{attribute 'qualified_only'}
{attribute 'strict'}
TYPE E_UserMgmtEventType :
(
	None := 0,
    UserCreated := 1,
    UserDeleted := 2,
    GroupUpdated := 3,
    AutoLogoutUpdated := 4,
    UserUpdated := 5,
    PasswordChanged := 6
);
END_TYPE

(* stored: Version 1.1.0.1, ProductVersion 3.1.4024.15
   DUT E_UserMgmtEventType: Id {1c1d8daf-4605-42b1-8235-e30080001eb9} *)
